{attribute 'linkalways'} 
{attribute 'no_explicit_call' := 'This FB is a CLASS and must be accessed using methods or properties'}
{attribute 'enable_dynamic_creation'}
FUNCTION_BLOCK _BOOL EXTENDS DatatypeBase
VAR
	localData : BOOL;
	activeData : REFERENCE TO BOOL REF= localData;
END_VAR

PROPERTY PUBLIC Address : PVOID
GET
Address := ADR(activeData);
END_GET
END_PROPERTY

METHOD PUBLIC ClearReference
VAR_INPUT
END_VAR
activeData REF= localData;
END_METHOD

METHOD PUBLIC Clone : I_Datatype
VAR
    pClone : POINTER TO _BOOL;
END_VAR
pClone := __NEW(_BOOL(InitialValue := Value));
Clone := pClone^;
END_METHOD

METHOD FB_init : BOOL
VAR_INPUT
	bInitRetains : BOOL; // if TRUE, the retain variables are initialized (warm start / cold start)
	bInCopyCode : BOOL;  // if TRUE, the instance afterwards gets moved into the copy code (online change)
	InitialValue : BOOL;
END_VAR
localData := InitialValue;
END_METHOD

METHOD PUBLIC MakeReferenceTo
VAR_INPUT
	ReferenceTarget : REFERENCE TO BOOL;
END_VAR
activeData REF= ReferenceTarget;
END_METHOD

METHOD PUBLIC SerializeWith
VAR_INPUT
	Serializer : I_Serializer;
END_VAR
Serializer.AddBool(activeData);
END_METHOD

PROPERTY PUBLIC Size : UDINT
GET
Size := SIZEOF(activeData);
END_GET
END_PROPERTY

METHOD TryDeserializeFrom : BOOL
VAR_INPUT
	Deserializer : I_Deserializer;
	Feedback : I_DeserializerFeedback;
END_VAR
TryDeserializeFrom := Deserializer.TryGetBool(activeData, Feedback);
END_METHOD

METHOD TryMakeReferenceTo : BOOL
VAR_INPUT
	Target : I_Datatype;
END_VAR
VAR
	pTargetData : POINTER TO BOOL;
END_VAR
IF NOT (Target.TypeName = TypeName) THEN
	RETURN;
END_IF

pTargetData := Target.Address;
activeData REF= pTargetData^;
TryMakeReferenceTo := TRUE;
END_METHOD

PROPERTY PUBLIC TypeName : T_MAXSTRING
GET
TypeName := 'BOOL';
END_GET
END_PROPERTY

PROPERTY PUBLIC Value : BOOL
GET
Value := activeData;
END_GET
SET
activeData := Value;
END_SET
END_PROPERTY

END_FUNCTION_BLOCK

(* stored: Version 1.1.0.1, ProductVersion 3.1.4024.12
   POU _BOOL: Id {eaa26018-a1d2-4691-aca3-616e2339c4b5}, SpecialFunc None
   Folder Constructor: Id {43c4b1fe-f90f-41f7-976e-393a7905dde0}
   Property Address: Id {db3770de-40d8-43af-ab2b-dc411369b4e1}
   Get Get: Id {cf7ea30f-d0ee-4aa6-ad6e-5d3fca25b886}
   Method ClearReference: Id {c5c6a5ae-1778-473a-beb0-c682456f8e68}
   Method Clone: Id {b5995843-029e-4631-b104-4b9f933442c5}
   Method FB_init: Id {f4865285-d74b-422f-bce5-6ef0c67c009e}
   Method MakeReferenceTo: Id {2246dab4-d526-485b-b191-fb980c693375}
   Method SerializeWith: Id {4ad6d86d-bf36-42e2-adb5-3c0e03736424}
   Property Size: Id {1acbc9cd-0eeb-46ab-8642-9a62c868285e}
   Get Get: Id {df8177a2-eb8b-4948-ae02-8c1cec5f9567}
   Method TryDeserializeFrom: Id {bdd5c23d-1e40-4a5f-8140-85d005da28f9}
   Method TryMakeReferenceTo: Id {99f568b7-bd08-4864-a8d9-726469a98320}
   Property TypeName: Id {9a4d08be-1111-4921-966c-60b74311e65a}
   Get Get: Id {17c8a9c0-cacd-492c-91df-18f518c756e0}
   Property Value: Id {cc6109a0-fa5c-4248-a615-127661da43a8}
   Get Get: Id {146293d5-64f8-40a4-bdf9-cc376c1205f9}
   Set Set: Id {2f2e43e8-def9-474d-8d8e-533c52110421} *)
